(* CODESYS project PLS1 Lekkasjedeteksjon 19.07.2021.ecp
   CompiledLibraryCompatibilityVersion: e!COCKPIT

Project tree, tasks and I/O mapping:
  Controller : 750-8213 PFC200 G2 2ETH CAN, WAGO, order no. 0750-8213, version 5.15.4.20
    application PLS1_Lekasje
      libraries: ; VisuDialogs, * (System); CmpEventMgr, 3.5.14.0 (System); Component Manager, 3.5.13.0 (System); CmpApp, 3.5.14.0 (System); CmpIecTask, 3.5.14.0 (System); WagoAppCloud, * (WAGO); WagoAppJSON, 1.1.0.13 (WAGO); WagoAppString, 1.6.3.1 (WAGO); WagoAppTime, 1.7.3.3 (WAGO)
      task PLC_Task (cyclic, interval 100 ms, priority 10, watchdog 90 ms x 1) calls PLC_PRG
      task MQTT (cyclic, interval 5000 ms, priority 15, watchdog 4500 ms x 1) calls Simulation_MQTT
      task VISU_TASK (cyclic, interval 200 ms, priority 15) calls VisuElems.Visu_Prg
      program PLC_PRG [ST]
      GlobalData/
        global variables HMI
        global variables IO
        global variables Local
        global variables SIM
        global variables STATUS
      program Alarms [ST]
      program Initialize [ST]
      program Inputs [ST]
      program Outputs [ST]
      program Simulation [ST]
      program Simulation_MQTT [ST]
      visualisation Visualization
      Symbols
      program Control [ST]
      global variables PersistentVars
      function RestartOpcUaMqttLinkOnDownload [ST]
      function RestartOpcUaMqttLinkOnOnlineChange [ST]
      Utils/
        data type OpcUa_Mqtt_Status
      LibHmiStructs/
        data type TestMcTestFace
        data type AlarmDigitalHmiCmd
        data type AlarmDigitalHmiPv
        data type AliveHmiPv
        data type PowerMonitoringHmiCmd
        data type PowerMonitoringHmiPv
        data type ScalingHmiCmd
        data type ScalingHmiPv
        data type SignalAnalogHmiCmd
        data type SignalAnalogHmiPv
        data type TimerHmiCmd
        data type TimerHmiPv
      LibFB/
        function block AlarmDigitalFB [ST]
        function block PowerMonitoringFb [ST]
        function block ScalingFB [ST]
        function block SignalAnalogFB [ST]
        function block TimerFB [ST]
    ProjectConfigurationTxt
    ProjectConfiguration
    Kbus : Kbus, WAGO, version 1.4.0.2
        unmapped channels: K-BUS diagnostics
      _4_DI_Generic : 075x-8DI, WAGO, order no. 075x-8DI, version 0.0.0.13
          settings: K-BUS Module slot index = 1
          unmapped channels: _IN
      _4AI_4_20mA_SE_T : 075x-8DO, WAGO, order no. 075x-8DO, version 0.0.0.13
          settings: K-BUS Module slot index = 2
          unmapped channels: _OUT
    MODBUS
      MODBUS : MODBUS, WAGO, order no. n/a, version 1.1.1.15
    CANbus
    Common.PCI
  text list GlobalTextList
  00000000-0000-0000-0000-000000000000|C:\Users\WagoNorgeLab-1\AppData\Local\Temp\d3cb062a7f514532819d4ea960a2affb\Project.xml
  00000000-0000-0000-0000-000000000000|C:\Users\WagoNorgeLab-1\AppData\Local\Temp\9d41c1f76f9443d88afca8bf8793c6d0\ProjectCfg.txt
  00000000-0000-0000-0000-000000000000|C:\Users\WagoNorgeLab-1\AppData\Local\Temp\27b794570e324c9d91450f12b7cda0c7\ProjectCfg.txt
  00000000-0000-0000-0000-000000000000|C:\Users\WagoNorgeLab-1\AppData\Local\Temp\8aecc143a5ab4543ad6828306d253df1\Project.xml
*)

// Controller/PLS1_Lekasje/LibHmiStructs/TestMcTestFace
TYPE TestMcTestFace :
STRUCT
	testString:STRING;
	testValue:INT:=0;
	testState:BOOL:=FALSE;
END_STRUCT
END_TYPE

// Controller/PLS1_Lekasje/Utils/OpcUa_Mqtt_Status
TYPE OpcUa_Mqtt_Status :
STRUCT
	LastRun:STRING;
	AliveCounterPv:INT := 0;
	Restart_Cmd:BOOL := FALSE;
END_STRUCT
END_TYPE

// Controller/PLS1_Lekasje/LibHmiStructs/AlarmDigitalHmiCmd
// These are autogenerated, do not manual modify it
TYPE AlarmDigitalHmiCmd :
STRUCT
	_tagId: STRING;
	_type: STRING;
	_owner: STRING;
	Tag:	STRING;
	Description:	STRING;
	Delay:	TimerHmiCmd;
	Acknowledged:	BOOL;
END_STRUCT
END_TYPE

// Controller/PLS1_Lekasje/LibHmiStructs/AlarmDigitalHmiPv
// These are autogenerated, do not manual modify it
TYPE AlarmDigitalHmiPv :
STRUCT
	_tagId: STRING;
	_type: STRING;
	_owner: STRING;
	Input_Pv:	BOOL;
	Delay:	TimerHmiPv;
	Alarm:	BOOL;
END_STRUCT
END_TYPE

// Controller/PLS1_Lekasje/LibHmiStructs/AliveHmiPv
TYPE AliveHmiPv :
STRUCT
	_tagId:STRING;
	_type: STRING;
	_owner: STRING;
	CounterPv:INT;
END_STRUCT
END_TYPE

// Controller/PLS1_Lekasje/LibHmiStructs/PowerMonitoringHmiCmd
//These are autogenerated, do not manual modify it
TYPE PowerMonitoringHmiCmd :
STRUCT
	_tagId: STRING;
	_type: STRING;
	_owner: STRING;
	BatterySize_Cmd:REAL; //Size of the battery in mAh
	
	
	
END_STRUCT
END_TYPE

// Controller/PLS1_Lekasje/LibHmiStructs/PowerMonitoringHmiPv
//These are autogenerated, do not manual modify it
TYPE PowerMonitoringHmiPv :
STRUCT
_tagId: STRING;
_type: STRING;
_owner: STRING;
Status_string:STRING;
Status_bool:BOOL;
Time_string:STRING;
Time_pv:REAL;
Alarm:BOOL;
Input_Current_In:REAL;
Input_Current_Out:REAL;
Input_Battery_Level:REAL;

END_STRUCT
END_TYPE

// Controller/PLS1_Lekasje/LibHmiStructs/ScalingHmiCmd
// These are autogenerated, do not manual modify it
TYPE ScalingHmiCmd :
STRUCT
	_tagId: STRING;
	_type: STRING;
	_owner: STRING;
	InputUnit:STRING;
	InputMin_Cmd:REAL;
	InputMax_Cmd:REAL;
	OutputUnit:STRING;
	OutputMin_Cmd:REAL;
	OutputMax_Cmd:REAL;
END_STRUCT
END_TYPE

// Controller/PLS1_Lekasje/LibHmiStructs/ScalingHmiPv
// These are autogenerated, do not manual modify it
TYPE ScalingHmiPv :
STRUCT
_tagId: STRING;
_type: STRING;
_owner: STRING;
Input_Pv:REAL;
Output_Pv:REAL;
END_STRUCT
END_TYPE

// Controller/PLS1_Lekasje/LibHmiStructs/SignalAnalogHmiCmd
// These are autogenerated, do not manual modify it
TYPE SignalAnalogHmiCmd :
STRUCT
_tagId: STRING;
_type: STRING;
_owner: STRING;
Tag:STRING;
Description:STRING;
AlarmHigh:AlarmDigitalHmiCmd;
AlarmHighHigh:AlarmDigitalHmiCmd;
AlarmLow:AlarmDigitalHmiCmd;
AlarmLowLow:AlarmDigitalHmiCmd;
AlarmHighLimit:REAL;
AlarmHighHighLimit:REAL;
AlarmLowLimit:REAL;
AlarmLowLowLimit:REAL;
AlarmHysteresis:REAL;
SimulationMode:BOOL;
SimulationValue:REAL;
InputScaling:ScalingHmiCmd;
END_STRUCT
END_TYPE

// Controller/PLS1_Lekasje/LibHmiStructs/SignalAnalogHmiPv
// These are autogenerated, do not manual modify it
TYPE SignalAnalogHmiPv :
STRUCT
_tagId: STRING;
_type: STRING;
_owner: STRING;
RawInput_Pv:REAL;
Output_Pv:REAL;
AlarmHigh:AlarmDigitalHmiPv;
AlarmHighHigh:AlarmDigitalHmiPv;
AlarmLow:AlarmDigitalHmiPv;
AlarmLowLow:AlarmDigitalHmiPv;
InputScaling:ScalingHmiPv;
END_STRUCT
END_TYPE

// Controller/PLS1_Lekasje/LibHmiStructs/TimerHmiCmd
// These are autogenerated, do not manual modify it
TYPE TimerHmiCmd :
STRUCT
	_tagId:STRING;
	_type: STRING;
	_owner: STRING;
	Tag:	STRING;
	Description:	STRING;
	OnDelayLimit:	REAL;
	OffDelayLimit:	REAL;
END_STRUCT
END_TYPE

// Controller/PLS1_Lekasje/LibHmiStructs/TimerHmiPv
// These are autogenerated, do not manual modify it
TYPE TimerHmiPv :
STRUCT
	_tagId:STRING;
	_type: STRING;
	_owner: STRING;
	Input_Pv:	BOOL;
	Output_Pv:	BOOL;
	OnDelayElapsed:	REAL;
	OffDelayElapsed:	REAL;
END_STRUCT
END_TYPE

// Controller/PLS1_Lekasje/GlobalData/HMI
{attribute 'qualified_only'}
VAR_GLOBAL PERSISTENT RETAIN
	
	FlowLevel1Cmd:SignalAnalogHmiCmd;
	FlowLevel2Cmd:SignalAnalogHmiCmd;
	FlowLevel3Cmd:SignalAnalogHmiCmd;
	FlowLevel4Cmd:SignalAnalogHmiCmd;
	FlowLevel5Cmd:SignalAnalogHmiCmd;
	FlowLevel6Cmd:SignalAnalogHmiCmd;
	FlowLevel7Cmd:SignalAnalogHmiCmd;
	
	BatteryMonitoring1Cmd:PowerMonitoringHmiCmd;
	BatteryMonitoring2Cmd:PowerMonitoringHmiCmd;
	BatteryMonitoring3Cmd:PowerMonitoringHmiCmd;
END_VAR

VAR_GLOBAL
	AliveCounterPlc1Pv:AliveHmiPv;
	AliveCounterTest:INT:=0;
	
	FlowLevel1Pv:SignalAnalogHmiPv;
	FlowLevel2Pv:SignalAnalogHmiPv;
	FlowLevel3Pv:SignalAnalogHmiPv;
	FlowLevel4Pv:SignalAnalogHmiPv;
	FlowLevel5Pv:SignalAnalogHmiPv;
	FlowLevel6Pv:SignalAnalogHmiPv;
	FlowLevel7Pv:SignalAnalogHmiPv;
	
	BatteryMonitoring1Pv:PowerMonitoringHmiPv;
	BatteryMonitoring2Pv:PowerMonitoringHmiPv;
	BatteryMonitoring3Pv:PowerMonitoringHmiPv;
	tester:TestMcTestFace;
	
END_VAR

// Controller/PLS1_Lekasje/GlobalData/IO
{attribute 'qualified_only'}
VAR_GLOBAL
	AI_FlowLevel1Pv:REAL;
	AI_FlowLevel2Pv:real;
	AI_FlowLevel3Pv:real;
	AI_FlowLevel4Pv:real;
	AI_FlowLevel5Pv:real;
	AI_FlowLevel6Pv:real;
	AI_FlowLevel7Pv:REAL;
	
	
	AI_CurrentIn01Pv :REAL;
	AI_CurentOut01Pv :REAL;
	AI_BatteryLevel01Pv :REAL;
	AI_CurrentIn02Pv :REAL;
	AI_CurentOut02Pv :REAL;
	AI_BatteryLevel02Pv :REAL;
	AI_CurrentIn03Pv :REAL;
	AI_CurentOut03Pv :REAL;
	AI_BatteryLevel03Pv :REAL;
END_VAR

// Controller/PLS1_Lekasje/GlobalData/Local
{attribute 'qualified_only'}
VAR_GLOBAL 
FlowLevel1:SignalAnalogFB;
FlowLevel2:SignalAnalogFB;
FlowLevel3:SignalAnalogFB;
FlowLevel4:SignalAnalogFB;
FlowLevel5:SignalAnalogFB;
FlowLevel6:SignalAnalogFB;
FlowLevel7:SignalAnalogFB;
BatteryMonitoring1 : PowerMonitoringFB;
BatteryMonitoring2 : PowerMonitoringFB;
BatteryMonitoring3 : PowerMonitoringFB;
END_VAR

// Controller/PLS1_Lekasje/GlobalData/SIM
{attribute 'qualified_only'}
VAR_GLOBAL
	WaterFlowFT01_Pv :REAL;
	WaterFlowFT02_Pv :REAL;
	WaterFlowFT03_Pv :REAL;
	WaterFlowFT04_Pv :REAL;
	WaterFlowFT05_Pv :REAL;
	WaterFlowFT06_Pv :REAL;
	WaterFlowFT07_Pv :REAL;
	CurrentIn01_Pv :REAL;
	CurentOut01_Pv :REAL;
	BatteryLevel01_Pv :REAL;
	CurrentIn02_Pv :REAL;
	CurentOut02_Pv :REAL;
	BatteryLevel02_Pv :REAL;
	CurrentIn03_Pv :REAL;
	CurentOut03_Pv :REAL;
	BatteryLevel03_Pv :REAL;
END_VAR

// Controller/PLS1_Lekasje/GlobalData/STATUS
{attribute 'qualified_only'}
VAR_GLOBAL
	OpcUaMqttLinkStatus: OpcUa_Mqtt_Status;
	
END_VAR

// Controller/PLS1_Lekasje/PersistentVars
{attribute 'qualified_only'}
VAR_GLOBAL PERSISTENT RETAIN
	
	
	// Generated instance path of persistent variable
	HMI.FlowLevel1Cmd: SignalAnalogHmiCmd;
	// Generated instance path of persistent variable
	HMI.FlowLevel2Cmd: SignalAnalogHmiCmd;
	// Generated instance path of persistent variable
	HMI.FlowLevel3Cmd: SignalAnalogHmiCmd;
	// Generated instance path of persistent variable
	HMI.FlowLevel4Cmd: SignalAnalogHmiCmd;
	// Generated instance path of persistent variable
	HMI.FlowLevel5Cmd: SignalAnalogHmiCmd;
	// Generated instance path of persistent variable
	HMI.FlowLevel6Cmd: SignalAnalogHmiCmd;
	// Generated instance path of persistent variable
	HMI.FlowLevel7Cmd: SignalAnalogHmiCmd;
	// Generated instance path of persistent variable
	HMI.BatteryMonitoring1Cmd: PowerMonitoringHmiCmd;
	// Generated instance path of persistent variable
	HMI.BatteryMonitoring2Cmd: PowerMonitoringHmiCmd;
	// Generated instance path of persistent variable
	HMI.BatteryMonitoring3Cmd: PowerMonitoringHmiCmd;
END_VAR

// Controller/PLS1_Lekasje/PLC_PRG
PROGRAM PLC_PRG
VAR
	_firstScan:BOOL := TRUE;
	_counter:INT;
	_lastRun:STRING;
END_VAR

// Signaling that the PLC is alive
Hmi.AliveCounterPlc1Pv._tagId := 'AliveCounterPlc1Pv';
Hmi.AliveCounterPlc1Pv._type := 'AliveHmi';
Hmi.AliveCounterPlc1Pv._owner := 'plc1';
HMI.AliveCounterPlc1Pv.CounterPv := HMI.AliveCounterPlc1Pv.CounterPv + 1;

_counter := STATUS.OpcUaMqttLinkStatus.AliveCounterPv;
_lastRun := STATUS.OpcUaMqttLinkStatus.LastRun;


IF _firstScan THEN
	Initialize();
END_IF
Inputs();
Alarms();
Control();
Outputs();
Simulation();



HMI.AliveCounterTest := HMI.AliveCounterTest +1;




// Always last
_firstScan := FALSE;

END_PROGRAM

// Controller/PLS1_Lekasje/Initialize
PROGRAM Initialize
VAR
END_VAR

HMI.BatteryMonitoring1Cmd.BatterySize_Cmd := 20;
HMI.BatteryMonitoring2Cmd.BatterySize_Cmd :=20;
HMI.BatteryMonitoring3Cmd.BatterySize_Cmd :=20;


Hmi.FlowLevel1Cmd.Tag := 'FT01';
Hmi.FlowLevel1Cmd.Description := 'Level of flow out of FT01';
Hmi.FlowLevel1Cmd.AlarmHysteresis := 10.0;
Hmi.FlowLevel1Cmd.AlarmHighHighLimit := 900.0;
Hmi.FlowLevel1Cmd.AlarmHighLimit := 800.0;
Hmi.FlowLevel1Cmd.AlarmLowLowLimit := 10.0;
Hmi.FlowLevel1Cmd.AlarmLowLimit := 20.0;
Hmi.FlowLevel1Cmd.AlarmHigh.Delay.OnDelayLimit := 1.0;
Hmi.FlowLevel1Cmd.AlarmHigh.Delay.OffDelayLimit := 1.0;
Hmi.FlowLevel1Cmd.AlarmHighHigh.Delay.OnDelayLimit := 1.0;
Hmi.FlowLevel1Cmd.AlarmHighHigh.Delay.OffDelayLimit := 1.0;
Hmi.FlowLevel1Cmd.AlarmLow.Delay.OnDelayLimit := 1.0;
Hmi.FlowLevel1Cmd.AlarmLow.Delay.OffDelayLimit := 1.0;
Hmi.FlowLevel1Cmd.AlarmLowLow.Delay.OnDelayLimit := 1.0;
Hmi.FlowLevel1Cmd.AlarmLowLow.Delay.OffDelayLimit := 1.0;
Hmi.FlowLevel1Cmd.InputScaling.InputUnit := 'na';
Hmi.FlowLevel1Cmd.InputScaling.OutputUnit := 'l/s';
Hmi.FlowLevel1Cmd.InputScaling.InputMax_Cmd := 100.0;
Hmi.FlowLevel1Cmd.InputScaling.InputMin_Cmd := 0.0;
Hmi.FlowLevel1Cmd.InputScaling.OutputMax_Cmd := 100.0;
Hmi.FlowLevel1Cmd.InputScaling.OutputMin_Cmd := 0.0;

Hmi.FlowLevel2Cmd.Tag := 'FT02';
Hmi.FlowLevel2Cmd.Description := 'Level of flow out of FT02';
Hmi.FlowLevel2Cmd.AlarmHysteresis := 10.0;
Hmi.FlowLevel2Cmd.AlarmHighHighLimit := 900.0;
Hmi.FlowLevel2Cmd.AlarmHighLimit := 800.0;
Hmi.FlowLevel2Cmd.AlarmLowLowLimit := 10.0;
Hmi.FlowLevel2Cmd.AlarmLowLimit := 20.0;
Hmi.FlowLevel2Cmd.AlarmHigh.Delay.OnDelayLimit := 1.0;
Hmi.FlowLevel2Cmd.AlarmHigh.Delay.OffDelayLimit := 1.0;
Hmi.FlowLevel2Cmd.AlarmHighHigh.Delay.OnDelayLimit := 1.0;
Hmi.FlowLevel2Cmd.AlarmHighHigh.Delay.OffDelayLimit := 1.0;
Hmi.FlowLevel2Cmd.AlarmLow.Delay.OnDelayLimit := 1.0;
Hmi.FlowLevel2Cmd.AlarmLow.Delay.OffDelayLimit := 1.0;
Hmi.FlowLevel2Cmd.AlarmLowLow.Delay.OnDelayLimit := 1.0;
Hmi.FlowLevel2Cmd.AlarmLowLow.Delay.OffDelayLimit := 1.0;
Hmi.FlowLevel2Cmd.InputScaling.InputUnit := 'na';
Hmi.FlowLevel2Cmd.InputScaling.OutputUnit := 'l/s';
Hmi.FlowLevel2Cmd.InputScaling.InputMax_Cmd := 100.0;
Hmi.FlowLevel2Cmd.InputScaling.InputMin_Cmd := 0.0;
Hmi.FlowLevel2Cmd.InputScaling.OutputMax_Cmd := 100.0;
Hmi.FlowLevel2Cmd.InputScaling.OutputMin_Cmd := 0.0;

Hmi.FlowLevel3Cmd.Tag := 'FT03';
Hmi.FlowLevel3Cmd.Description := 'Level of flow out of FT03';
Hmi.FlowLevel3Cmd.AlarmHysteresis := 10.0;
Hmi.FlowLevel3Cmd.AlarmHighHighLimit := 900.0;
Hmi.FlowLevel3Cmd.AlarmHighLimit := 800.0;
Hmi.FlowLevel3Cmd.AlarmLowLowLimit := 10.0;
Hmi.FlowLevel3Cmd.AlarmLowLimit := 20.0;
Hmi.FlowLevel3Cmd.AlarmHigh.Delay.OnDelayLimit := 1.0;
Hmi.FlowLevel3Cmd.AlarmHigh.Delay.OffDelayLimit := 1.0;
Hmi.FlowLevel3Cmd.AlarmHighHigh.Delay.OnDelayLimit := 1.0;
Hmi.FlowLevel3Cmd.AlarmHighHigh.Delay.OffDelayLimit := 1.0;
Hmi.FlowLevel3Cmd.AlarmLow.Delay.OnDelayLimit := 1.0;
Hmi.FlowLevel3Cmd.AlarmLow.Delay.OffDelayLimit := 1.0;
Hmi.FlowLevel3Cmd.AlarmLowLow.Delay.OnDelayLimit := 1.0;
Hmi.FlowLevel3Cmd.AlarmLowLow.Delay.OffDelayLimit := 1.0;
Hmi.FlowLevel3Cmd.InputScaling.InputUnit := 'na';
Hmi.FlowLevel3Cmd.InputScaling.OutputUnit := 'l/s';
Hmi.FlowLevel3Cmd.InputScaling.InputMax_Cmd := 100.0;
Hmi.FlowLevel3Cmd.InputScaling.InputMin_Cmd := 0.0;
Hmi.FlowLevel3Cmd.InputScaling.OutputMax_Cmd := 100.0;
Hmi.FlowLevel3Cmd.InputScaling.OutputMin_Cmd := 0.0;

Hmi.FlowLevel4Cmd.Tag := 'FT04';
Hmi.FlowLevel4Cmd.Description := 'Level of flow out of FT04';
Hmi.FlowLevel4Cmd.AlarmHysteresis := 10.0;
Hmi.FlowLevel4Cmd.AlarmHighHighLimit := 900.0;
Hmi.FlowLevel4Cmd.AlarmHighLimit := 800.0;
Hmi.FlowLevel4Cmd.AlarmLowLowLimit := 10.0;
Hmi.FlowLevel4Cmd.AlarmLowLimit := 20.0;
Hmi.FlowLevel4Cmd.AlarmHigh.Delay.OnDelayLimit := 1.0;
Hmi.FlowLevel4Cmd.AlarmHigh.Delay.OffDelayLimit := 1.0;
Hmi.FlowLevel4Cmd.AlarmHighHigh.Delay.OnDelayLimit := 1.0;
Hmi.FlowLevel4Cmd.AlarmHighHigh.Delay.OffDelayLimit := 1.0;
Hmi.FlowLevel4Cmd.AlarmLow.Delay.OnDelayLimit := 1.0;
Hmi.FlowLevel4Cmd.AlarmLow.Delay.OffDelayLimit := 1.0;
Hmi.FlowLevel4Cmd.AlarmLowLow.Delay.OnDelayLimit := 1.0;
Hmi.FlowLevel4Cmd.AlarmLowLow.Delay.OffDelayLimit := 1.0;
Hmi.FlowLevel4Cmd.InputScaling.InputUnit := 'na';
Hmi.FlowLevel4Cmd.InputScaling.OutputUnit := 'l/s';
Hmi.FlowLevel4Cmd.InputScaling.InputMax_Cmd := 100.0;
Hmi.FlowLevel4Cmd.InputScaling.InputMin_Cmd := 0.0;
Hmi.FlowLevel4Cmd.InputScaling.OutputMax_Cmd := 100.0;
Hmi.FlowLevel4Cmd.InputScaling.OutputMin_Cmd := 0.0;

Hmi.FlowLevel5Cmd.Tag := 'FT05';
Hmi.FlowLevel5Cmd.Description := 'Level of flow out of FT05';
Hmi.FlowLevel5Cmd.AlarmHysteresis := 10.0;
Hmi.FlowLevel5Cmd.AlarmHighHighLimit := 900.0;
Hmi.FlowLevel5Cmd.AlarmHighLimit := 800.0;
Hmi.FlowLevel5Cmd.AlarmLowLowLimit := 10.0;
Hmi.FlowLevel5Cmd.AlarmLowLimit := 20.0;
Hmi.FlowLevel5Cmd.AlarmHigh.Delay.OnDelayLimit := 1.0;
Hmi.FlowLevel5Cmd.AlarmHigh.Delay.OffDelayLimit := 1.0;
Hmi.FlowLevel5Cmd.AlarmHighHigh.Delay.OnDelayLimit := 1.0;
Hmi.FlowLevel5Cmd.AlarmHighHigh.Delay.OffDelayLimit := 1.0;
Hmi.FlowLevel5Cmd.AlarmLow.Delay.OnDelayLimit := 1.0;
Hmi.FlowLevel5Cmd.AlarmLow.Delay.OffDelayLimit := 1.0;
Hmi.FlowLevel5Cmd.AlarmLowLow.Delay.OnDelayLimit := 1.0;
Hmi.FlowLevel5Cmd.AlarmLowLow.Delay.OffDelayLimit := 1.0;
Hmi.FlowLevel5Cmd.InputScaling.InputUnit := 'na';
Hmi.FlowLevel5Cmd.InputScaling.OutputUnit := 'l/s';
Hmi.FlowLevel5Cmd.InputScaling.InputMax_Cmd := 100.0;
Hmi.FlowLevel5Cmd.InputScaling.InputMin_Cmd := 0.0;
Hmi.FlowLevel5Cmd.InputScaling.OutputMax_Cmd := 100.0;
Hmi.FlowLevel5Cmd.InputScaling.OutputMin_Cmd := 0.0;

Hmi.FlowLevel6Cmd.Tag := 'FT06';
Hmi.FlowLevel6Cmd.Description := 'Level of flow out of FT06';
Hmi.FlowLevel6Cmd.AlarmHysteresis := 10.0;
Hmi.FlowLevel6Cmd.AlarmHighHighLimit := 900.0;
Hmi.FlowLevel6Cmd.AlarmHighLimit := 800.0;
Hmi.FlowLevel6Cmd.AlarmLowLowLimit := 10.0;
Hmi.FlowLevel6Cmd.AlarmLowLimit := 20.0;
Hmi.FlowLevel6Cmd.AlarmHigh.Delay.OnDelayLimit := 1.0;
Hmi.FlowLevel6Cmd.AlarmHigh.Delay.OffDelayLimit := 1.0;
Hmi.FlowLevel6Cmd.AlarmHighHigh.Delay.OnDelayLimit := 1.0;
Hmi.FlowLevel6Cmd.AlarmHighHigh.Delay.OffDelayLimit := 1.0;
Hmi.FlowLevel6Cmd.AlarmLow.Delay.OnDelayLimit := 1.0;
Hmi.FlowLevel6Cmd.AlarmLow.Delay.OffDelayLimit := 1.0;
Hmi.FlowLevel6Cmd.AlarmLowLow.Delay.OnDelayLimit := 1.0;
Hmi.FlowLevel6Cmd.AlarmLowLow.Delay.OffDelayLimit := 1.0;
Hmi.FlowLevel6Cmd.InputScaling.InputUnit := 'na';
Hmi.FlowLevel6Cmd.InputScaling.OutputUnit := 'l/s';
Hmi.FlowLevel6Cmd.InputScaling.InputMax_Cmd := 100.0;
Hmi.FlowLevel6Cmd.InputScaling.InputMin_Cmd := 0.0;
Hmi.FlowLevel6Cmd.InputScaling.OutputMax_Cmd := 100.0;
Hmi.FlowLevel6Cmd.InputScaling.OutputMin_Cmd := 0.0;

Hmi.FlowLevel7Cmd.Tag := 'FT07';
Hmi.FlowLevel7Cmd.Description := 'Level of flow out of FT07';
Hmi.FlowLevel7Cmd.AlarmHysteresis := 10.0;
Hmi.FlowLevel7Cmd.AlarmHighHighLimit := 900.0;
Hmi.FlowLevel7Cmd.AlarmHighLimit := 800.0;
Hmi.FlowLevel7Cmd.AlarmLowLowLimit := 10.0;
Hmi.FlowLevel7Cmd.AlarmLowLimit := 20.0;
Hmi.FlowLevel7Cmd.AlarmHigh.Delay.OnDelayLimit := 1.0;
Hmi.FlowLevel7Cmd.AlarmHigh.Delay.OffDelayLimit := 1.0;
Hmi.FlowLevel7Cmd.AlarmHighHigh.Delay.OnDelayLimit := 1.0;
Hmi.FlowLevel7Cmd.AlarmHighHigh.Delay.OffDelayLimit := 1.0;
Hmi.FlowLevel7Cmd.AlarmLow.Delay.OnDelayLimit := 1.0;
Hmi.FlowLevel7Cmd.AlarmLow.Delay.OffDelayLimit := 1.0;
Hmi.FlowLevel7Cmd.AlarmLowLow.Delay.OnDelayLimit := 1.0;
Hmi.FlowLevel7Cmd.AlarmLowLow.Delay.OffDelayLimit := 1.0;
Hmi.FlowLevel7Cmd.InputScaling.InputUnit := 'na';
Hmi.FlowLevel7Cmd.InputScaling.OutputUnit := 'l/s';
Hmi.FlowLevel7Cmd.InputScaling.InputMax_Cmd := 100.0;
Hmi.FlowLevel7Cmd.InputScaling.InputMin_Cmd := 0.0;
Hmi.FlowLevel7Cmd.InputScaling.OutputMax_Cmd := 100.0;
Hmi.FlowLevel7Cmd.InputScaling.OutputMin_Cmd := 0.0;

END_PROGRAM

// Controller/PLS1_Lekasje/Inputs
PROGRAM Inputs
VAR
END_VAR



Local.FlowLevel1(_id := 'FlowLevel1', _owner := 'plc1',
				RawInput := IO.AI_FlowLevel1Pv,
				HmiCmd := HMI.FlowLevel1Cmd,
				HmiPv := HMI.FlowLevel1Pv);	
	
Local.FlowLevel2(_id := 'FlowLevel2', _owner := 'plc1',
				RawInput := IO.AI_FlowLevel2Pv,
				HmiCmd := HMI.FlowLevel2Cmd,
				HmiPv := HMI.FlowLevel2Pv);

Local.FlowLevel3(_id := 'FlowLevel3', _owner := 'plc1',
				RawInput := IO.AI_FlowLevel3Pv,
				HmiCmd := HMI.FlowLevel3Cmd,
				HmiPv := HMI.FlowLevel3Pv);		
	
Local.FlowLevel4(_id := 'FlowLevel4', _owner := 'plc1',
				RawInput := IO.AI_FlowLevel4Pv,
				HmiCmd := HMI.FlowLevel4Cmd,
				HmiPv := HMI.FlowLevel4Pv);		

Local.FlowLevel5(_id := 'FlowLevel5', _owner := 'plc1',
				RawInput := IO.AI_FlowLevel5Pv,
				HmiCmd := HMI.FlowLevel5Cmd,
				HmiPv := HMI.FlowLevel5Pv);		

Local.FlowLevel6(_id := 'FlowLevel6', _owner := 'plc1',
				RawInput := IO.AI_FlowLevel6Pv,
				HmiCmd := HMI.FlowLevel6Cmd,
				HmiPv := HMI.FlowLevel6Pv);		

Local.FlowLevel7(_id := 'FlowLevel7', _owner := 'plc1',
				RawInput := IO.AI_FlowLevel7Pv,
				HmiCmd := HMI.FlowLevel7Cmd,
				HmiPv := HMI.FlowLevel7Pv);

END_PROGRAM

// Controller/PLS1_Lekasje/Alarms
PROGRAM Alarms
VAR
END_VAR

END_PROGRAM

// Controller/PLS1_Lekasje/Control
PROGRAM Control
VAR
END_VAR



Local.BatteryMonitoring1(_id:= 'BatteryMonitoring1', 	_owner:= 'plc1', 
	Input_CurrentIn:=IO.AI_CurrentIn01Pv , 
	Input_CurrentOut:= IO.AI_CurentOut01Pv, 
	Input_CurrentStored:= IO.AI_BatteryLevel01Pv, 
	HmiCmd:= HMI.BatteryMonitoring1Cmd, 
	HmiPv:=HMI.BatteryMonitoring1Pv );
	
Local.BatteryMonitoring2(_id:= 'BatteryMonitoring2', 	_owner:= 'plc1', 
	Input_CurrentIn:=IO.AI_CurrentIn02Pv , 
	Input_CurrentOut:= IO.AI_CurentOut02Pv, 
	Input_CurrentStored:= IO.AI_BatteryLevel02Pv, 
	HmiCmd:= HMI.BatteryMonitoring2Cmd, 
	HmiPv:=HMI.BatteryMonitoring2Pv );
	
Local.BatteryMonitoring3(_id:= 'BatteryMonitoring3', 	_owner:= 'plc1', 
	Input_CurrentIn:=IO.AI_CurrentIn03Pv , 
	Input_CurrentOut:= IO.AI_CurentOut03Pv, 
	Input_CurrentStored:= IO.AI_BatteryLevel03Pv, 
	HmiCmd:= HMI.BatteryMonitoring3Cmd, 
	HmiPv:=HMI.BatteryMonitoring3Pv );

END_PROGRAM

// Controller/PLS1_Lekasje/Outputs
PROGRAM Outputs
VAR
END_VAR

END_PROGRAM

// Controller/PLS1_Lekasje/Simulation
PROGRAM Simulation
VAR
END_VAR

// Simulation because no physical IO is connected
IO.AI_FlowLevel1Pv := SIM.WaterFlowFT01_Pv;
IO.AI_FlowLevel2Pv := SIM.WaterFlowFT02_Pv;
IO.AI_FlowLevel3Pv := SIM.WaterFlowFT03_Pv;
IO.AI_FlowLevel4Pv := SIM.WaterFlowFT04_Pv;
IO.AI_FlowLevel5Pv := SIM.WaterFlowFT05_Pv;
IO.AI_FlowLevel6Pv := SIM.WaterFlowFT06_Pv;
IO.AI_FlowLevel7Pv := SIM.WaterFlowFT07_Pv;

IO.AI_CurrentIn01Pv := SIM.CurrentIn01_Pv;
IO.AI_CurentOut01Pv := SIM.CurentOut01_Pv;
IO.AI_BatteryLevel01Pv :=SIM.BatteryLevel01_Pv;
IO.AI_CurrentIn02Pv := SIM.CurrentIn02_Pv;
IO.AI_CurentOut02Pv := SIM.CurentOut02_Pv;
IO.AI_BatteryLevel02Pv :=SIM.BatteryLevel02_Pv;
IO.AI_CurrentIn03Pv := SIM.CurrentIn03_Pv;
IO.AI_CurentOut03Pv := SIM.CurentOut03_Pv;
IO.AI_BatteryLevel03Pv :=SIM.BatteryLevel03_Pv;

END_PROGRAM

// Controller/PLS1_Lekasje/Simulation_MQTT
PROGRAM Simulation_MQTT
VAR
	MqttStatus 				: WagoAppCloud.FbStatus_NativeMQTT;
	MqttError				: BOOL := FALSE;
	MqttConnectedToMyCloud	: BOOL := FALSE;
	MqttFillLevel			: REAL := 0;
	MqttOutgoingBlocks		: ULINT := 0;
	
	
	
	MqttSubscribe 				: WagoAppCloud.FbSubscribeMQTT;
	MqttSubscriptionDataBytes	: ARRAY [0..512] OF BYTE;
	MqttSubscriptionDataJSONString			: STRING(JSON_MAX_STRING);	//	Resulting JSON string
	MqttSubscriptionDataJSONPointer			: WagoAppJSON.typJSON_Pointer;
	MqttSubcriptionJSONParser				: Fb_JSON_ParseAndModify;	//	JSON parser function block
	MqttSubscribeNewData: BOOL;
	
	oParserStatus	: WagoAppJSON.WagoSysErrorBase.FbResult;
	xParserError	: BOOL;
	xParserDone		: BOOL;
	diParserToken	: DINT;
	xParserBuildup	: BOOL;
	xParserTrigger	: ARRAY[0..15] OF BOOL;
	
	MqttPublish 		: WagoAppCloud.FbPublishMQTT;
	MqttPublishParameters	: ARRAY[0..10] OF STRING;
	MqttPublishTemplate		: STRING(512) := '{"#Parameter": #Parameter}';
	JSONWriter 		: FB_JSON_Writer_01;
	MqttPublishPayload		: STRING(1024);
	MqttPublishBuffer			: ARRAY[0..1999] OF BYTE;
	MqttPublishTrigger : BOOL;
	JSONWriter_Done	: BOOL;
	JSONWriter_Error	: BOOL;
	JSONWriter_Status		: WagoSysErrorBase.FbResult;
	JSONWriterTrigger	: BOOL;
END_VAR

// Status
MqttStatus(xEnabled := TRUE,
		   xError => MqttError,
		   xCloudConnected => MqttConnectedToMyCloud,			// Will be FALSE after network timeout occured 
		   rCacheFillLevel => MqttFillLevel,					// Increasing value indicates bad network or overload
		   uliOutgoingDataBlocks => MqttOutgoingBlocks);  	// Only for QoS 1 and 2. Increasing value indicates bad network or overload
		   
// Subscribe to data		   
MqttSubscribe(xSubscribe := TRUE, 
	sTopic := 'ba/wago/sim/plc1/plcsub', 
	eQoS := eQualityOfService.QoS1, 
	aPayloadData:= MqttSubscriptionDataBytes,
	xDataReceived => MqttSubscribeNewData);

MemCopySecure(pDest:= ADR(MqttSubscriptionDataJSONString), udiDestSize:= 255, pSource:= ADR(MqttSubscriptionDataBytes), udiSourceSize:= MqttSubscribe.dwRxNBytes, bPadding:= 0);

//	Execute this function block once to complete the parser buildup process
//	This must be done before calling the parser methods

IF MqttSubscribeNewData THEN
	xParserBuildup := TRUE;
END_IF

MqttSubcriptionJSONParser(
	pData:= ADR(MqttSubscriptionDataJSONString), 			//	JSON string to parse
	udiSizeData:= length(MqttSubscriptionDataJSONString), 
	oStatus=> oParserStatus, 
	xError=> xParserError, 
	xDone=> xParserDone, 
	diToken=> diParserToken, 
	xTrigger:= xParserBuildup);		//	Set xParserBuildup TRUE to execute the function block
	
IF xParserDone THEN
	xParserTrigger[0] := TRUE;			//	Set xParserTrigger TRUE to execute the parser method
	xParserTrigger[1] := TRUE;			
	xParserTrigger[2] := TRUE;			
	xParserTrigger[3] := TRUE;
	xParserTrigger[4] := TRUE;
	xParserTrigger[5] := TRUE;	
	xParserTrigger[6] := TRUE;	
	xParserTrigger[7] := TRUE;	
	xParserTrigger[8] := TRUE;	
	xParserTrigger[9] := TRUE;	
	xParserTrigger[10] := TRUE;	
	xParserTrigger[11] := TRUE;	
	xParserTrigger[12] := TRUE;	
	xParserTrigger[13] := TRUE;	
	xParserTrigger[14] := TRUE;	
	xParserTrigger[15] := TRUE;			
	xParserDone := FALSE;
END_IF

//	Call the parser method GetValueByPath for each value to be extracted from the JSON string
MqttSubscriptionDataJSONPointer := MqttSubcriptionJSONParser.GetValueByPath(sPointer:='/FT01',xTrigger:=xParserTrigger[0]);
SIM.WaterFlowFT01_Pv := STRING_TO_REAL(MqttSubscriptionDataJSONPointer.sValue);

MqttSubscriptionDataJSONPointer := MqttSubcriptionJSONParser.GetValueByPath(sPointer:='/FT02',xTrigger:=xParserTrigger[1]);
SIM.WaterFlowFT02_Pv := STRING_TO_REAL(MqttSubscriptionDataJSONPointer.sValue);

MqttSubscriptionDataJSONPointer := MqttSubcriptionJSONParser.GetValueByPath(sPointer:='/FT03',xTrigger:=xParserTrigger[2]);
SIM.WaterFlowFT03_Pv := STRING_TO_REAL(MqttSubscriptionDataJSONPointer.sValue);

MqttSubscriptionDataJSONPointer := MqttSubcriptionJSONParser.GetValueByPath(sPointer:='/FT04',xTrigger:=xParserTrigger[3]);
SIM.WaterFlowFT04_Pv := STRING_TO_REAL(MqttSubscriptionDataJSONPointer.sValue);

MqttSubscriptionDataJSONPointer := MqttSubcriptionJSONParser.GetValueByPath(sPointer:='/FT05',xTrigger:=xParserTrigger[4]);
SIM.WaterFlowFT05_Pv := STRING_TO_REAL(MqttSubscriptionDataJSONPointer.sValue);

MqttSubscriptionDataJSONPointer := MqttSubcriptionJSONParser.GetValueByPath(sPointer:='/FT06',xTrigger:=xParserTrigger[5]);
SIM.WaterFlowFT06_Pv := STRING_TO_REAL(MqttSubscriptionDataJSONPointer.sValue);

MqttSubscriptionDataJSONPointer := MqttSubcriptionJSONParser.GetValueByPath(sPointer:='/FT07',xTrigger:=xParserTrigger[6]);
SIM.WaterFlowFT07_Pv := STRING_TO_REAL(MqttSubscriptionDataJSONPointer.sValue);

MqttSubscriptionDataJSONPointer := MqttSubcriptionJSONParser.GetValueByPath(sPointer:='/CI01',xTrigger:=xParserTrigger[7]);
SIM.CurrentIn01_Pv := STRING_TO_REAL(MqttSubscriptionDataJSONPointer.sValue);

MqttSubscriptionDataJSONPointer := MqttSubcriptionJSONParser.GetValueByPath(sPointer:='/CO01',xTrigger:=xParserTrigger[8]);
SIM.CurentOut01_Pv := STRING_TO_REAL(MqttSubscriptionDataJSONPointer.sValue);

MqttSubscriptionDataJSONPointer := MqttSubcriptionJSONParser.GetValueByPath(sPointer:='/BL01',xTrigger:=xParserTrigger[9]);
SIM.BatteryLevel01_Pv := STRING_TO_REAL(MqttSubscriptionDataJSONPointer.sValue);

MqttSubscriptionDataJSONPointer := MqttSubcriptionJSONParser.GetValueByPath(sPointer:='/CI02',xTrigger:=xParserTrigger[10]);
SIM.CurrentIn02_Pv := STRING_TO_REAL(MqttSubscriptionDataJSONPointer.sValue);

MqttSubscriptionDataJSONPointer := MqttSubcriptionJSONParser.GetValueByPath(sPointer:='/CO02',xTrigger:=xParserTrigger[11]);
SIM.CurentOut02_Pv := STRING_TO_REAL(MqttSubscriptionDataJSONPointer.sValue);

MqttSubscriptionDataJSONPointer := MqttSubcriptionJSONParser.GetValueByPath(sPointer:='/BL02',xTrigger:=xParserTrigger[12]);
SIM.BatteryLevel02_Pv := STRING_TO_REAL(MqttSubscriptionDataJSONPointer.sValue);

MqttSubscriptionDataJSONPointer := MqttSubcriptionJSONParser.GetValueByPath(sPointer:='/CI03',xTrigger:=xParserTrigger[13]);
SIM.CurrentIn03_Pv := STRING_TO_REAL(MqttSubscriptionDataJSONPointer.sValue);

MqttSubscriptionDataJSONPointer := MqttSubcriptionJSONParser.GetValueByPath(sPointer:='/CO03',xTrigger:=xParserTrigger[14]);
SIM.CurentOut03_Pv := STRING_TO_REAL(MqttSubscriptionDataJSONPointer.sValue);

MqttSubscriptionDataJSONPointer := MqttSubcriptionJSONParser.GetValueByPath(sPointer:='/BL03',xTrigger:=xParserTrigger[15]);
SIM.BatteryLevel03_Pv := STRING_TO_REAL(MqttSubscriptionDataJSONPointer.sValue);

END_PROGRAM

// Controller/PLS1_Lekasje/RestartOpcUaMqttLinkOnDownload
FUNCTION RestartOpcUaMqttLinkOnDownload : DWORD
VAR_IN_OUT
	EventPrm: CmpApp.EVTPARAM_CmpApp;
END_VAR
VAR
END_VAR

(*
This function is called whan a download is about to happen. 
This will force the Opc Ua - MQTT link to restart.
The restart will take 10 seconds, allowing e!Cockpit to download and start before the link starts.
*)
Status.OpcUaMqttLinkStatus.Restart_Cmd := TRUE;

END_FUNCTION

// Controller/PLS1_Lekasje/RestartOpcUaMqttLinkOnOnlineChange
FUNCTION RestartOpcUaMqttLinkOnOnlineChange : DWORD
VAR_IN_OUT
	EventPrm: CmpApp.EVTPARAM_CmpApp;
END_VAR
VAR
END_VAR

(*
This function is called whan a online change is about to happen. 
This will force the Opc Ua - MQTT link to restart.
The restart will take 10 seconds, allowing e!Cockpit to download and start before the link starts.
*)
Status.OpcUaMqttLinkStatus.Restart_Cmd := TRUE;

END_FUNCTION

// Controller/PLS1_Lekasje/LibFB/AlarmDigitalFB
FUNCTION_BLOCK AlarmDigitalFB
VAR_INPUT
	_id:STRING;
	_owner:STRING;
	Input:	BOOL;
END_VAR
VAR_OUTPUT
	Alarm:	BOOL;
END_VAR
VAR
	_Delay:	TimerFB;
	_AlarmLastScan:BOOL;
	_type:string := 'AlarmDigital';
END_VAR
VAR_IN_OUT
	HmiCmd:	AlarmDigitalHmiCmd;
	HmiPv:	AlarmDigitalHmiPv;
END_VAR

(*
Name: AlarmDigitalFB
Author: Jone Vassbø
Version: 0.3
Date: 09.03.2020
Description:
- Function block for a digital alarm, with commands from HMI in seperate struct
*)

// In routine - start -
// Validate input
// In routine - end -
// Alarm routine - start
// Alarm routine - end -

// Control routine - start -
_Delay(_id := _id, _owner := _owner, Input := Input, Output => Alarm, HmiCmd := HmiCmd.Delay, HmiPv := HmiPv.Delay);
IF Alarm AND NOT _AlarmLastScan THEN // Flank
	HmiCmd.Acknowledged := FALSE;
END_IF
_AlarmLastScan := Alarm;
// Control routine - end -

// Out routine - start - 
HmiPv.Input_Pv := Input;
HmiPv.Alarm := Alarm OR NOT HmiCmd.Acknowledged;
HmiCmd._tagId := CONCAT(_id, 'Cmd');
HmiPv._tagId := CONCAT(_id, 'Pv');
HmiPv._type := _type;
HmiCmd._type := _type;
HmiPv._owner := _owner;
HmiCmd._owner := _owner;
// Out routine - end -

END_FUNCTION_BLOCK

// Controller/PLS1_Lekasje/LibFB/TimerFB
FUNCTION_BLOCK TimerFB
VAR_INPUT
	_id:STRING;
	_owner:STRING;
	Input:	BOOL;
END_VAR
VAR_OUTPUT
	Output:	BOOL;
END_VAR
VAR
	OnDelay: TON;
	OffDelay: TOF;
	ToSec:REAL := 1000.0;
	_type:string := 'Timer';
END_VAR
VAR_IN_OUT
	HmiCmd:	TimerHmiCmd;
	HmiPv: TimerHmiPv;
END_VAR

(*
Name: TimerFB
Author: Jone Vassbø
Version: 0.4
Date: 09.03.2020
Description:
- Function block operating as a Timer with both on and off delay
*)

// In routine - start -
// Validate input
IF HmiCmd.OnDelayLimit < 0 THEN
	HmiCmd.OnDelayLimit := 0.0;
END_IF
IF HmiCmd.OffDelayLimit < 0 THEN
	HmiCmd.OnDelayLimit := 0.0;
END_IF
// In routine - end -
// Alarm routine - start
// Alarm routine - end -
// Control routine - start -
OnDelay(IN := Input,
	PT := TO_TIME(HmiCmd.OnDelayLimit*ToSec));
HmiPv.OnDelayElapsed := TO_REAL(OnDelay.ET)/ToSec;

OffDelay(IN := OnDelay.Q,
	PT := TO_TIME(HmiCmd.OffDelayLimit*ToSec));
HmiPv.OffDelayElapsed := TO_REAL(OffDelay.ET)/ToSec;

IF OnDelay.Q THEN
	Output := TRUE;
END_IF
IF NOT OffDelay.Q THEN
	Output := FALSE;
END_IF
// Control routine - end -

// Out routine - start - 
HmiPv.Input_Pv := Input;
HmiPv.Output_Pv := Output;
HmiCmd._tagId := CONCAT(_id, 'Cmd');
HmiPv._tagId := CONCAT(_id, 'Pv');
HmiPv._type := _type;
HmiCmd._type := _type;
HmiPv._owner := _owner;
HmiCmd._owner := _owner;
// Out routine - end -

END_FUNCTION_BLOCK

// Controller/PLS1_Lekasje/LibFB/PowerMonitoringFb
FUNCTION_BLOCK PowerMonitoringFb
VAR_INPUT
	_id:STRING;
	_owner:STRING;
	Input_CurrentIn:REAL;
	Input_CurrentOut:REAL;
	Input_CurrentStored:REAL;
END_VAR
VAR_OUTPUT
END_VAR
VAR
	_type:STRING:= 'PowerMonitoring';
	Current_balance :REAL;
END_VAR
VAR_IN_OUT
	HmiCmd:PowerMonitoringHmiCmd;
	HmiPv:PowerMonitoringHmiPv;
END_VAR

(*
Name: PowerMonitoringFB
Author: Markus Raudberget
Version: 0.1
Date: 14.03.2020
Description:
- Function block for Power monitoring of a battery package, with commands from hmi i seperate struct
*)

//Control routine - start -
Current_balance := (Input_currentIn - Input_CurrentOut);
IF Current_balance <0 THEN
	HmiPv.Status_bool :=FALSE;
	HmiPv.Status_string :='Decharging';
	HmiPv.Time_pv := Input_CurrentStored / -Current_balance;
	HmiPv.Time_string :='Time for empty battery';
ELSE 
	HmiPv.Status_bool :=TRUE;
	HmiPv.Status_string :='Charging';
	HmiPv.Time_pv := (HmiCmd.BatterySize_Cmd - Input_CurrentStored) / Current_balance;
	HmiPv.Time_string :='Time for full battery';
END_IF

HmiPv.Input_Current_In :=Input_CurrentIn;
HmiPv.Input_Current_Out :=Input_CurrentOut;
HmiPv.Input_Battery_Level :=Input_CurrentStored;

HmiCmd._tagId := CONCAT(_id, 'Cmd');
HmiPv._tagId := CONCAT(_id, 'Pv');
HmiPv._type := _type;
HmiCmd._type := _type;
HmiPv._owner := _owner;
HmiCmd._owner := _owner;

END_FUNCTION_BLOCK

// Controller/PLS1_Lekasje/LibFB/ScalingFB
FUNCTION_BLOCK ScalingFB
VAR_INPUT
	_id:STRING;
	_owner:STRING;
	Input:REAL;
END_VAR
VAR_OUTPUT
	Output:REAL;
END_VAR
VAR
	_type:string := 'Scaling';
END_VAR
VAR_IN_OUT
	HmiCmd:ScalingHmiCmd;
	HmiPv:ScalingHmiPv;
END_VAR


(*
Name: ScalingFB
Author: Jone Vassbø
Version: 0.3
Date: 09.03.2020
Description:
- Function block for a scaling analog value, with commands from HMI in seperate struct
*)

// Control routine - start -
Output :=  HmiCmd.OutputMin_Cmd * (1 - ((Input - HmiCmd.InputMin_Cmd) / (HmiCmd.InputMax_Cmd - HmiCmd.InputMin_Cmd))) + HmiCmd.OutputMax_Cmd * ((Input - HmiCmd.InputMin_Cmd) / (HmiCmd.InputMax_Cmd - HmiCmd.InputMin_Cmd));
// Control routine - end -

// Out routine - start - 
HmiPv.Input_Pv := Input;
HmiPv.Output_Pv := Output;
HmiCmd._tagId := CONCAT(_id, 'Cmd');
HmiPv._tagId := CONCAT(_id, 'Pv');
HmiPv._type := _type;
HmiCmd._type := _type;
HmiCmd._owner := _owner;
HmiPv._owner := _owner;
// Out routine - end -

END_FUNCTION_BLOCK

// Controller/PLS1_Lekasje/LibFB/SignalAnalogFB
FUNCTION_BLOCK SignalAnalogFB
VAR_INPUT
	_id:STRING;
	_owner:STRING;
	RawInput:REAL;
END_VAR
VAR_OUTPUT
	Output:REAL;
	AlarmHigh:BOOL;
	AlarmHighHigh:BOOL;
	AlarmLow:BOOL;
	AlarmLowLow:BOOL;
END_VAR
VAR
	_AlarmHigh: AlarmDigitalFB;
	_AlarmHighHigh: AlarmDigitalFB;
	_AlarmLow: AlarmDigitalFB;
	_AlarmLowLow: AlarmDigitalFB;
	_Scaling: ScalingFB;
	
	_High:BOOL;
	_HighHigh:BOOL;
	_Low:BOOL;
	_LowLow:BOOL;
	
	_type:string := 'SignalAnalog';
END_VAR
VAR_IN_OUT
	HmiCmd:SignalAnalogHmiCmd;
	HmiPv:SignalAnalogHmiPv;
END_VAR

(*
Name: SignalAnalogFB
Author: Jone Vassbø
Version: 0.3
Date: 09.03.2020
Description:
- Function block for a analog signal, with alarms and commands from HMI in seperate struct
*)

// In routine - start -
// Validate input
_Scaling(_id := _id, _owner := _owner, Input:= RawInput, HmiCmd := HmiCmd.InputScaling, HmiPv := HmiPv.InputScaling);
IF HmiCmd.SimulationMode THEN
	Output := HmiCmd.SimulationValue;
ELSE
	Output := _Scaling.Output;
END_IF
// In routine - end -
// Alarm routine - start
IF Output > HmiCmd.AlarmHighLimit THEN
	_High := TRUE;
END_IF
IF Output < (HmiCmd.AlarmHighLimit - HmiCmd.AlarmHysteresis) THEN
	_High := FALSE;
END_IF
_AlarmHigh(_id := _id, _owner := _owner, Input :=  _High,
	HmiCmd := HmiCmd.AlarmHigh, HmiPv := HmiPv.AlarmHigh);

IF Output > HmiCmd.AlarmHighHighLimit THEN
	_HighHigh := TRUE;
END_IF
IF Output < (HmiCmd.AlarmHighHighLimit - HmiCmd.AlarmHysteresis) THEN
	_HighHigh := FALSE;
END_IF
_AlarmHighHigh(_id := _id, _owner := _owner, Input :=  _HighHigh,
	HmiCmd := HmiCmd.AlarmHighHigh, HmiPv := HmiPv.AlarmHighHigh);

IF Output < HmiCmd.AlarmLowLimit THEN
	_Low := TRUE;
END_IF
IF Output > (HmiCmd.AlarmLowLimit + HmiCmd.AlarmHysteresis) THEN
	_Low := FALSE;
END_IF
_AlarmLow(_id := _id, _owner := _owner, Input :=  _Low,
	HmiCmd := HmiCmd.AlarmLow, HmiPv := HmiPv.AlarmLow);
	
IF Output < HmiCmd.AlarmLowLowLimit THEN
	_LowLow := TRUE;
END_IF
IF Output > (HmiCmd.AlarmLowLowLimit + HmiCmd.AlarmHysteresis) THEN
	_LowLow := FALSE;
END_IF
_AlarmLowLow(_id := _id, _owner := _owner, Input :=  _LowLow,
	HmiCmd := HmiCmd.AlarmLowLow, HmiPv := HmiPv.AlarmLowLow);
// Alarm routine - end -

// Control routine - start -

// Control routine - end -

// Out routine - start - 
AlarmHigh := _AlarmHigh.Alarm OR NOT HmiCmd.AlarmHigh.Acknowledged;
AlarmHighHigh := _AlarmHighHigh.Alarm OR NOT HmiCmd.AlarmHighHigh.Acknowledged;
AlarmLow := _AlarmLow.Alarm OR NOT HmiCmd.AlarmLow.Acknowledged;
AlarmLowLow := _AlarmLowLow.Alarm OR NOT HmiCmd.AlarmLowLow.Acknowledged;

HmiPv.Output_Pv := Output;
HmiPv.RawInput_Pv := RawInput;
HmiCmd._tagId := CONCAT(_id, 'Cmd');
HmiPv._tagId := CONCAT(_id, 'Pv');
HmiPv._type := _type;
HmiCmd._type := _type;
HmiPv._owner := _owner;
HmiCmd._owner := _owner;
// Out routine - end -

END_FUNCTION_BLOCK

// Controller/PLS1_Lekasje/Visualization
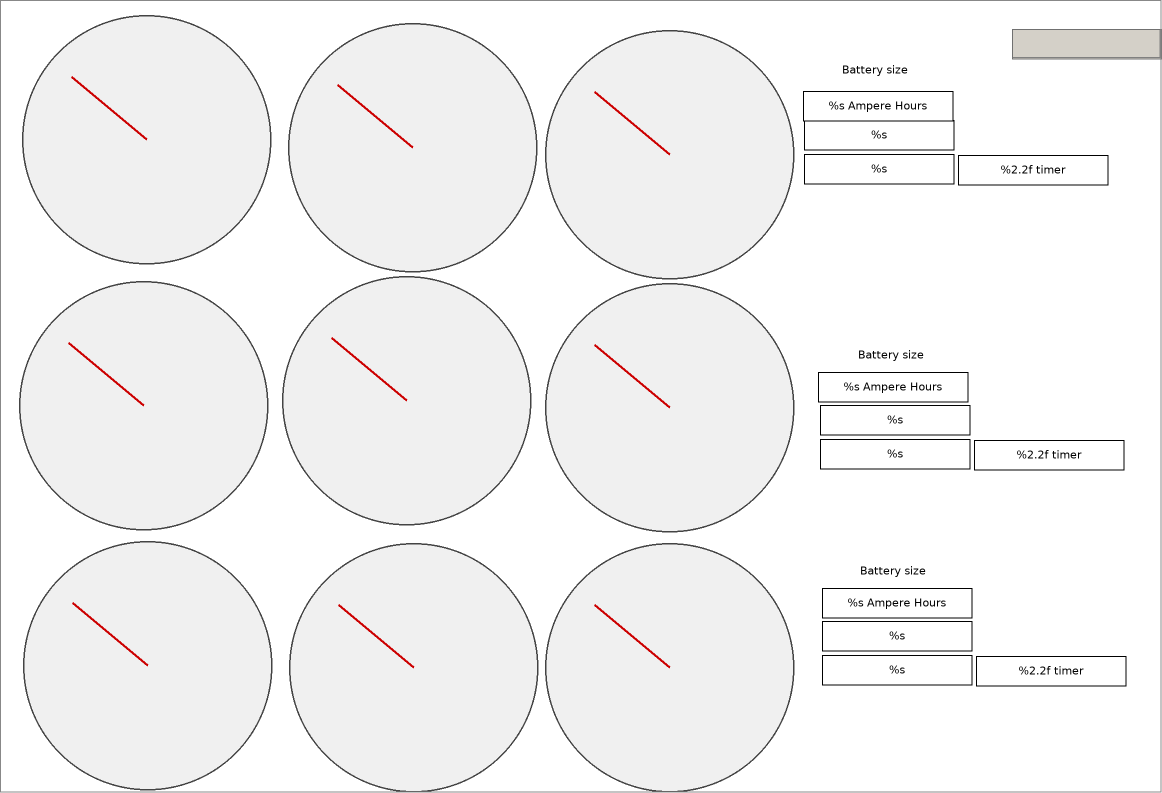
VISUALIZATION Visualization  // 1162x793
    Button (1012,29 150x30)
    Label (408,519 150x30), invisible if: HMI.BatteryMonitoring1Pv.Status_bool
    Meter360 (545,30 249x249), value: HMI.BatteryMonitoring1Pv.Input_Battery_Level, style: Meter-Meter360-Gray, scale format: %.1f, scale 0..20
        p518627256: Stored energy [Ah]
    Meter360 (22,15 249x249), value: HMI.BatteryMonitoring1Pv.Input_Current_In, style: Meter-Meter360-Gray, scale format: %.1f, scale 0..20
        p518627256: Current inn [A]
    Meter360 (288,23 249x249), value: HMI.BatteryMonitoring1Pv.Input_Current_Out, style: Meter-Meter360-Gray, scale format: %.1f, scale 0..10
        p518627256: Current out [A]
    Rectangle (804,120 150x30), "%s", text variable: HMI.BatteryMonitoring1Pv.Status_string
    Rectangle (804,154 150x30), "%s", text variable: HMI.BatteryMonitoring1Pv.Time_string
    Rectangle (803,91 150x30), "%s Ampere Hours", text variable: HMI.BatteryMonitoring1Cmd.BatterySize_Cmd
        OnMouseClick: write HMI.BatteryMonitoring1Cmd.BatterySize_Cmd via Default, min 0, max 100
    Label (800,55 150x30), "Battery size"
    Rectangle (958,155 150x30), "%2.2f timer", text variable: HMI.BatteryMonitoring1Pv.Time_pv
    Meter360 (19,281 249x249), value: HMI.BatteryMonitoring2Pv.Input_Current_In, style: Meter-Meter360-Gray, scale format: %.1f, scale 0..20
        p518627256: Current inn [A]
    Meter360 (23,541 249x249), value: HMI.BatteryMonitoring3Pv.Input_Current_In, style: Meter-Meter360-Gray, scale format: %.1f, scale 0..20
        p518627256: Current inn [A]
    Meter360 (282,276 249x249), value: HMI.BatteryMonitoring2Pv.Input_Current_Out, style: Meter-Meter360-Gray, scale format: %.1f, scale 0..10
        p518627256: Current out [A]
    Meter360 (289,543 249x249), value: HMI.BatteryMonitoring3Pv.Input_Current_Out, style: Meter-Meter360-Gray, scale format: %.1f, scale 0..10
        p518627256: Current out [A]
    Meter360 (545,283 249x249), value: HMI.BatteryMonitoring2Pv.Input_Battery_Level, style: Meter-Meter360-Gray, scale format: %.1f, scale 0..20
        p518627256: Stored energy [Ah]
    Meter360 (545,543 249x249), value: HMI.BatteryMonitoring3Pv.Input_Battery_Level, style: Meter-Meter360-Gray, scale format: %.1f, scale 0..20
        p518627256: Stored energy [Ah]
    Rectangle (822,621 150x30), "%s", text variable: HMI.BatteryMonitoring3Pv.Status_string
    Rectangle (822,655 150x30), "%s", text variable: HMI.BatteryMonitoring3Pv.Time_string
    Label (818,556 150x30), "Battery size"
    Rectangle (976,656 150x30), "%2.2f timer", text variable: HMI.BatteryMonitoring3Pv.Time_pv
    Rectangle (820,405 150x30), "%s", text variable: HMI.BatteryMonitoring2Pv.Status_string
    Rectangle (820,439 150x30), "%s", text variable: HMI.BatteryMonitoring2Pv.Time_string
    Label (816,340 150x30), "Battery size"
    Rectangle (974,440 150x30), "%2.2f timer", text variable: HMI.BatteryMonitoring2Pv.Time_pv
    Rectangle (818,372 150x30), "%s Ampere Hours", text variable: HMI.BatteryMonitoring2Cmd.BatterySize_Cmd
        OnMouseClick: write HMI.BatteryMonitoring2Cmd.BatterySize_Cmd via Default, min 0, max 20
    Rectangle (822,588 150x30), "%s Ampere Hours", text variable: HMI.BatteryMonitoring3Cmd.BatterySize_Cmd
        OnMouseClick: write HMI.BatteryMonitoring3Cmd.BatterySize_Cmd via Default, min 0, max 20
END_VISUALIZATION
